PROGRAM MAIN
VAR
	_state :UINT;
	actual_job : REFERENCE TO FB_Executor;
	executor: FB_Executor; // main Executor
	
	_child_executor : REFERENCE TO FB_Executor;
	
	task_blink_1 : FutureTimerBlink;
	task_blink_2 : FutureTimerBlink;
	task_count_1 : FutureCounterBlink;
	task_count_2 : FutureCounterBlink;

	future_counter_creator : FutureCounterBlinkCreator;
	future_timer_creator : FutureTimerBlinkCreator;

	
	component1_in : BOOL;
	component1_out : BOOL;
	component2_in : BOOL;
	component2_out : BOOL;
	component3_in : BOOL;
	component3_out : BOOL;
	component4_in : BOOL;
	component4_out : BOOL;

	
	// Dynamic instance use
	_future: InterfaceFuture;
	_container : InterfaceContainer;
	
	job_create_switch : ARRAY[1..4] OF BOOL;
	execution_step: STRING;
	resume: BOOL;
	abort: BOOL;
	reset : BOOL;
	task_info : __SYSTEM.VAR_INFO;
	
	fbObserver : FB_observer;
	fbJobTreeSearch : FB_ExecutorTreeSearch;
	
	end_of_manual: BOOL;
	init :BOOL;
	test_executor : POINTER TO FB_BatchJobContainer;
	
	future_timer : FutureTimerBlink;
	future_counter : FutureCounterBlink;
	
	_monitor_job : REFERENCE TO FB_Executor;
	_monitor_count_blinker : POINTER TO FutureCounterBlink;
	_monitor_time_blinker : POINTER TO FutureTimerBlink;
	
	_job_debug_monitoring : FB_Executor;
	
END_VAR

IF NOT init THEN
	//executor.job_event_reporter := fbObserver;
	init := TRUE;
	executor.id := 'ROOT';
	executor.upstream_aborting := FALSE;
	executor.create_container(ContainerType.PARALLEL_QUEUE,'BASE');
	executor.continuous_mode := TRUE;
	executor.Subscribe(fbObserver);
	//actual_job REF= executor.children.create_container(ContainerType.QUEUE, 'Batch Container');
	//actual_job.continuous_mode := TRUE;
END_IF

IF abort THEN
	executor.abort();
END_IF

executor.execute();

IF executor.ready THEN
	executor.start();
END_IF

IF resume THEN
	IF executor.error_reset() THEN
		IF executor.resume() THEN
			resume := FALSE;
		END_IF
	END_IF
END_IF



CASE _state OF
	0:
		_child_executor REF= executor.children.create_container(ContainerType.PARALLEL_QUEUE, 'Parallel Container');
		// Static instances
		task_blink_1.set_parameter(T#5S, component1_out);
		task_blink_1.future_name := 'Button 1 blink';
		task_blink_2.set_parameter(T#3S, component2_out);
		task_blink_2.future_name := 'Button 2 blink';
		task_count_1.set_parameter(3, component3_in,component3_out);
		task_count_1.future_name := 'Button 3 count';
		task_count_2.set_parameter(5, component4_in, component4_out);
		task_count_2.error_test := FALSE;
		task_count_2.future_name := 'Button 4 count';
		
		_child_executor.children.spawn_job(task_blink_1);
		_child_executor.children.spawn_job(task_blink_2);
		_child_executor.children.spawn_job(task_count_1);
		_child_executor.children.spawn_job(task_count_2);
		__QUERYPOINTER(_child_executor.children,test_executor);
		
		// dynamic instances		
		//_child_executor REF= actual_job.children.create_container(ContainerType.PARALLEL, 'Dynamic parallel tasks');
		
		future_counter_creator.set_parameter(2, component3_in, component3_out);
		_child_executor.children.create_job(future_counter_creator, 'Dynamic job : Count-1');	
		
		future_counter_creator.set_parameter(5, component4_in, component4_out);
		_child_executor.children.create_job(future_counter_creator, 'Dynamic job : Count-2');

		future_counter_creator.set_parameter(2,component3_in, component3_out);
		_child_executor.children.create_job(future_counter_creator, 'Dynamic job : Counter3');

		future_counter_creator.set_parameter(2, component3_in, component3_out);
		_child_executor.children.create_job(future_counter_creator, 'Dynamic job : Counter4'); // 同時実行でなければ同じFutureオブジェクトを使いまわせる
		future_counter_creator.set_parameter(2, component4_in, component4_out);
		_child_executor.children.create_job(future_counter_creator, 'Dynamic job : Counter5');
		
		// Report 'executor' job directory
		fbJobTreeSearch.subscriber := fbObserver;
		fbJobTreeSearch.search(executor);
			
		_state := 1;
	1:
		// シーケンス制御
		IF _child_executor.done THEN
			_state := 3;
		END_IF
	2:
		_state := 3;			
	3:
		
		IF job_create_switch[1] THEN
			future_timer_creator.set_parameter(T#5S, component1_out);
			future_timer_creator.set_options(FALSE);
			_monitor_job REF= executor.children.create_job(future_timer_creator, 'Button 1 Time blink 5s');
			IF NOT  __QUERYPOINTER(_monitor_job.future, _monitor_count_blinker) THEN
				_monitor_count_blinker := 0;
			END_IF
			IF NOT __QUERYPOINTER(_monitor_job.future, _monitor_time_blinker)  THEN
				_monitor_time_blinker := 0;
			END_IF
			job_create_switch[1] := FALSE;
		
		ELSIF job_create_switch[2] THEN
			future_timer_creator.set_parameter(T#3S, component2_out);
			future_timer_creator.set_options(FALSE);
			_monitor_job REF= executor.children.create_job(future_timer_creator, 'Button 2 Time blink 3s');
			IF NOT  __QUERYPOINTER(_monitor_job.future, _monitor_count_blinker) THEN
				_monitor_count_blinker := 0;
			END_IF
			IF NOT __QUERYPOINTER(_monitor_job.future, _monitor_time_blinker)  THEN
				_monitor_time_blinker := 0;
			END_IF
			job_create_switch[2] := FALSE;
		
		ELSIF  job_create_switch[3] THEN
			job_create_switch[3] := FALSE;
			future_counter_creator.set_parameter(2, component3_in, component3_out);
			future_counter_creator.set_options(FALSE);
			_monitor_job REF= executor.children.create_job(future_counter_creator, 'Dynamic job : Counter6');
			IF NOT  __QUERYPOINTER(_monitor_job.future, _monitor_count_blinker) THEN
				_monitor_count_blinker := 0;
			END_IF
			IF NOT __QUERYPOINTER(_monitor_job.future, _monitor_time_blinker)  THEN
				_monitor_time_blinker := 0;
			END_IF
			job_create_switch[3] := FALSE;
		ELSIF  job_create_switch[4] THEN
			job_create_switch[4] := FALSE;
			future_counter_creator.set_parameter(4, component4_in, component4_out);
			future_counter_creator.set_options(TRUE);
			_monitor_job REF= executor.children.create_job(future_counter_creator, 'Dynamic job : Counter7');
			IF NOT  __QUERYPOINTER(_monitor_job.future, _monitor_count_blinker) THEN
				_monitor_count_blinker := 0;
			END_IF
			IF NOT __QUERYPOINTER(_monitor_job.future, _monitor_time_blinker)  THEN
				_monitor_time_blinker := 0;
			END_IF
			job_create_switch[4] := FALSE;
		
		END_IF
		IF reset THEN
			executor.quit();
			_state := 4;
		END_IF
	4:
		_state := 0;
		
END_CASE

MEMCPY(ADR(_job_debug_monitoring), ADR(_child_executor), SIZEOF(_job_debug_monitoring));

IF reset AND NOT executor.busy THEN
	IF executor.children.reset(TRUE) THEN
		reset := FALSE;
	END_IF
END_IF

END_PROGRAM

(* stored: Version 1.1.0.1, ProductVersion 3.1.4024.12
   POU MAIN: Id {0711fc19-ddf5-4c28-b96d-7cde88b1723f}, SpecialFunc None *)
